FUNCTION func_f1: DINT
VAR_INPUT
    farg_f1_x: DINT;
END_VAR

func_f1 := (farg_f1_x) + (1);
RETURN;

END_FUNCTION

(* stored: ProductVersion 3.1.0.18, Version 1.1.0.1 *)
